(* LS Electric XG5000 project: 엘리베이터 프로젝트(내부 구현) *)
(* PLC LSPLC *)
(* module base 0 slot 0: FEnet:XGL-EFMT(B) (Fast Ethernet 통신 모듈, 전기 Master) *)
(* module base 0 slot 1: 입력 모듈:XGI-D21A (DC 24V 입력, 8점 (전류소스/싱크입력)) *)
(* module base 0 slot 2: 출력 모듈:XGQ-RY1A (릴레이 출력, 8점 (2A용, 단독 COM.)) *)
(* task 초기화: Kind=1 Priority=2 *)
VAR_GLOBAL
    ADD : INT;
    D0 : INT;
    D1 : INT;
    SUB : INT;
    열림TP : TP;
    타이머1 : TON;
END_VAR

(* Comments on direct variables
%MX0	상승
%MX1	하강
%MX2	문 열림
%MX3	문 닫힘
%MX4	도착
%MX5	비상 사태
%MX6	LOCK
%MX20	현재 1층 위치
%MX21	현재 2층 위치
%MX22	현재 3층 위치
%MX23	현재 4층 위치
%MX24	현재 5층 위치
%MX100	내부 1층 버튼
%MX101	내부2층버튼
%MX102	내부3층 버튼
%MX103	내부4층버튼
%MX104	내부5층버튼
%MX105	문열림 버튼
%MX106	문닫힘버튼
%MX107	외부1층상승
%MX108	외부 2층상승
%MX109	외부2층하강
%MX110	외부3층상승
%MX111	외부3층하강
%MX112	외부4층상승
%MX113	외부4층하강
%MX114	외부5층하강
%QX0.2.0	1층 램프
%QX0.2.1	2층 램프
%QX0.2.2	3층 램프
%QX0.2.3	4층 램프
%QX0.2.4	5층 램프
%QX0.2.5	문 열림
%QX0.2.6	문 닫힘
*)

PROGRAM 내부 (* task: 스캔 프로그램 *)
VAR_EXTERNAL
    D0 : INT;
    D1 : INT;
END_VAR
VAR
    D10 : INT;
    T2 : TON;
END_VAR
VAR
    _e1 : R_TRIG;
    _e2 : R_TRIG;
    _e3 : R_TRIG;
    _e4 : R_TRIG;
    _e5 : R_TRIG;
    _e6 : R_TRIG;
    _e7 : R_TRIG;
    _e8 : R_TRIG;
    _e9 : R_TRIG;
    _e10 : R_TRIG;
    _e11 : R_TRIG;
    _e12 : R_TRIG;
    _e13 : R_TRIG;
    _t14 : BOOL;
END_VAR

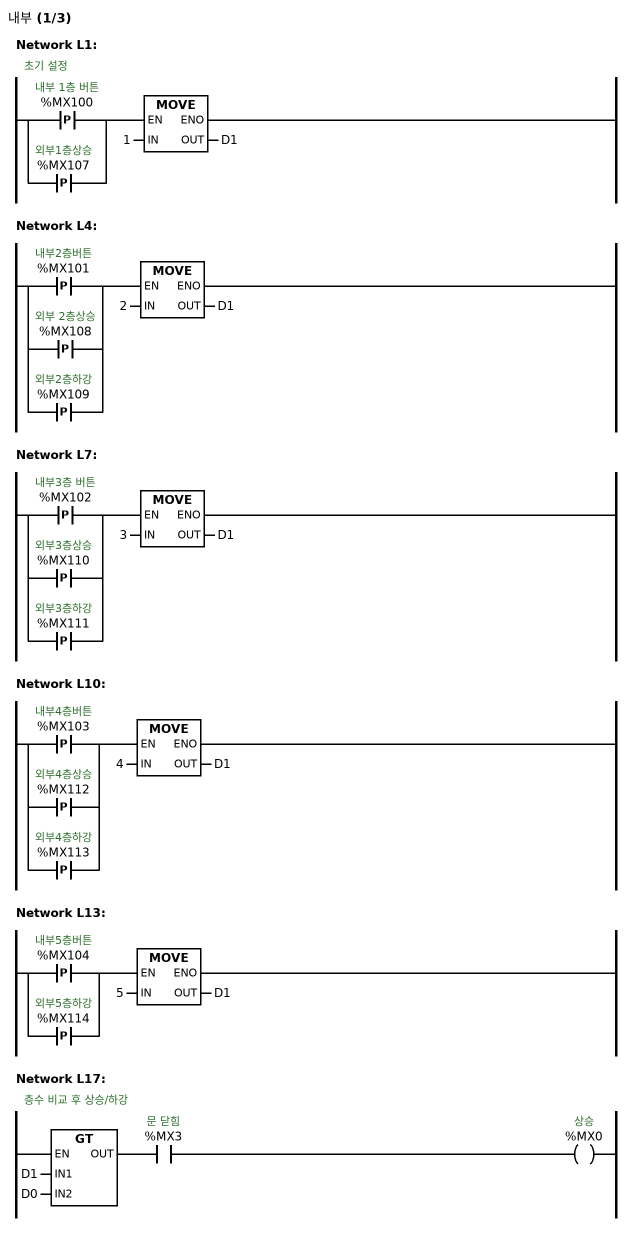
(* 초기 설정 *)
(* Rung L1 *)
_e1(CLK := %MX100);
_e2(CLK := %MX107);
IF _e1.Q OR _e2.Q THEN D1 := 1; END_IF;
(* Rung L4 *)
_e3(CLK := %MX101);
_e4(CLK := %MX108);
_e5(CLK := %MX109);
IF _e3.Q OR _e4.Q OR _e5.Q THEN D1 := 2; END_IF;
(* Rung L7 *)
_e6(CLK := %MX102);
_e7(CLK := %MX110);
_e8(CLK := %MX111);
IF _e6.Q OR _e7.Q OR _e8.Q THEN D1 := 3; END_IF;
(* Rung L10 *)
_e9(CLK := %MX103);
_e10(CLK := %MX112);
_e11(CLK := %MX113);
IF _e9.Q OR _e10.Q OR _e11.Q THEN D1 := 4; END_IF;
(* Rung L13 *)
_e12(CLK := %MX104);
_e13(CLK := %MX114);
IF _e12.Q OR _e13.Q THEN D1 := 5; END_IF;
(* 층수 비교 후 상승/하강 *)
(* Rung L17 *)
%MX0 := (D1 > D0) AND %MX3;

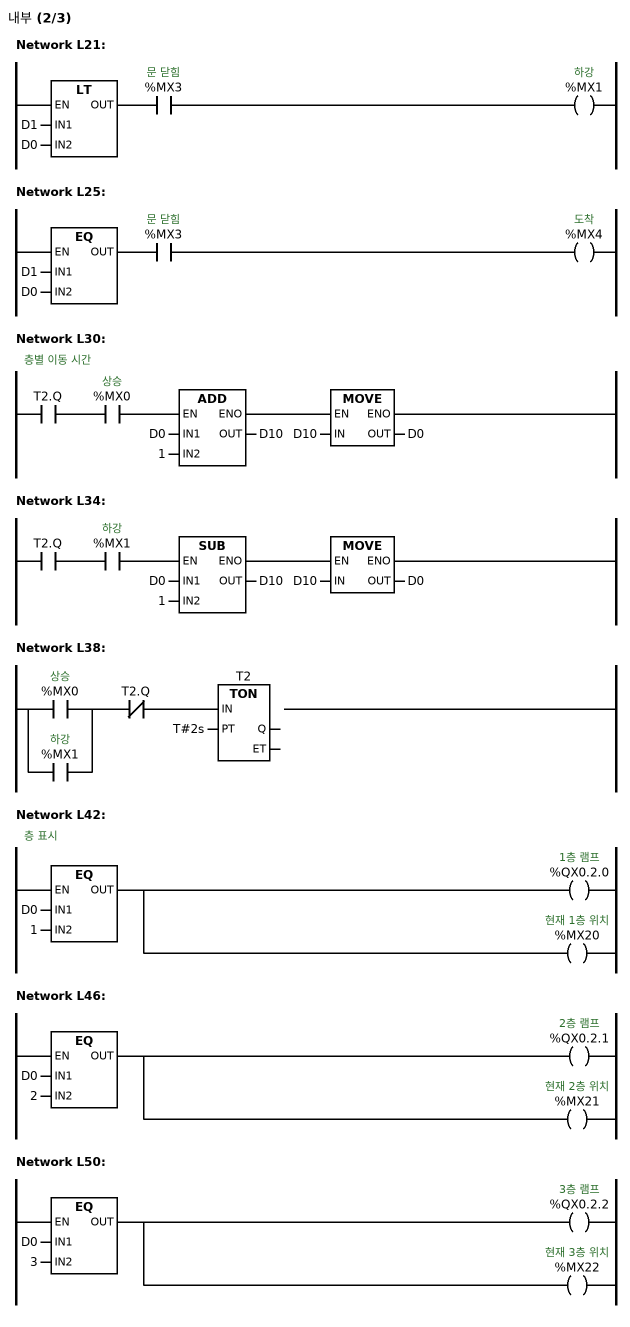
(* Rung L21 *)
%MX1 := (D1 < D0) AND %MX3;
(* Rung L25 *)
%MX4 := (D1 = D0) AND %MX3;
(* 층별 이동 시간 *)
(* Rung L30 *)
IF T2.Q AND %MX0 THEN
    D10 := D0 + 1;
    D0 := D10;
END_IF;
(* Rung L34 *)
IF T2.Q AND %MX1 THEN
    D10 := D0 - 1;
    D0 := D10;
END_IF;
(* Rung L38 *)
T2(IN := (%MX0 OR %MX1) AND NOT T2.Q, PT := T#2s);
(* 층 표시 *)
(* Rung L42 *)
%QX0.2.0 := D0 = 1;
%MX20 := D0 = 1;
(* Rung L46 *)
%QX0.2.1 := D0 = 2;
%MX21 := D0 = 2;
(* Rung L50 *)
%QX0.2.2 := D0 = 3;
%MX22 := D0 = 3;

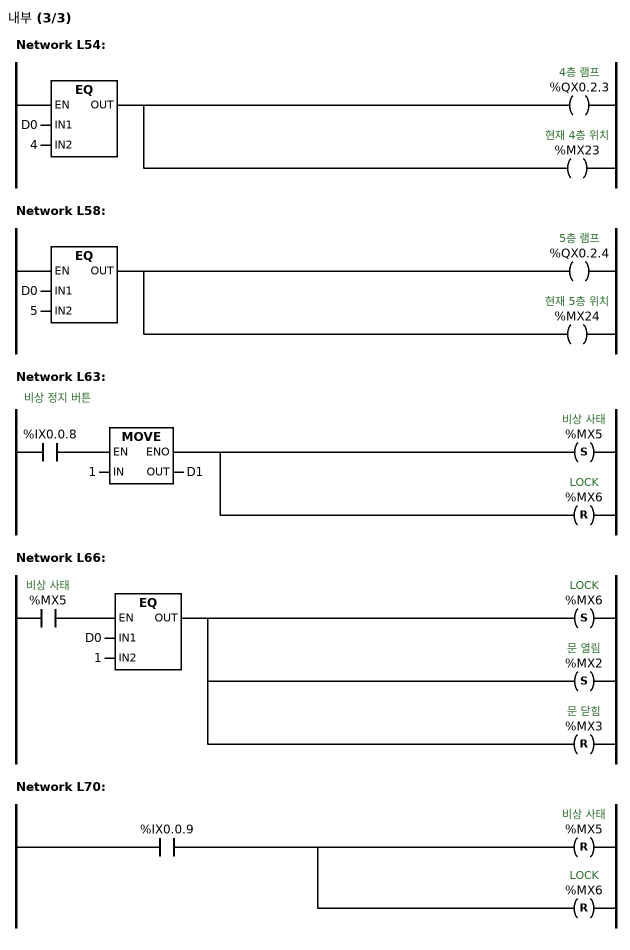
(* Rung L54 *)
%QX0.2.3 := D0 = 4;
%MX23 := D0 = 4;
(* Rung L58 *)
%QX0.2.4 := D0 = 5;
%MX24 := D0 = 5;
(* 비상 정지 버튼 *)
(* Rung L63 *)
IF %IX0.0.8 THEN
    D1 := 1;
    %MX5 := TRUE;
    %MX6 := FALSE;
END_IF;
(* Rung L66 *)
IF %MX5 THEN _t14 := D0 = 1; END_IF;
IF _t14 THEN
    %MX6 := TRUE;
    %MX2 := TRUE;
    %MX3 := FALSE;
END_IF;
(* Rung L70 *)
IF %IX0.0.9 THEN
    %MX5 := FALSE;
    %MX6 := FALSE;
END_IF;
END_PROGRAM

PROGRAM Timer (* task: 스캔 프로그램 *)
VAR
    CTU1 : CTU_INT;
    CTU2 : CTU_INT;
    D0 : SINT;
    OPEN : TP;
    T1 : TON;
    T2 : TON;
END_VAR
VAR_EXTERNAL
    열림TP : TP;
    타이머1 : TON;
END_VAR

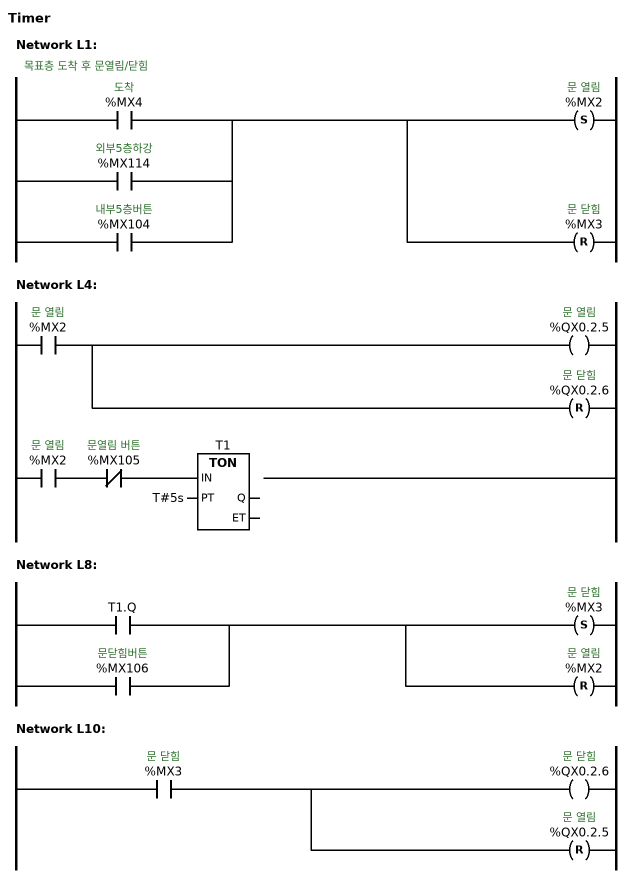
(* 목표층 도착 후 문열림/닫힘 *)
(* Rung L1 *)
IF %MX4 OR %MX114 OR %MX104 THEN
    %MX2 := TRUE;
    %MX3 := FALSE;
END_IF;
(* Rung L4 *)
%QX0.2.5 := %MX2;
IF %MX2 THEN %QX0.2.6 := FALSE; END_IF;
T1(IN := %MX2 AND NOT %MX105, PT := T#5s);
(* Rung L8 *)
IF T1.Q OR %MX106 THEN
    %MX3 := TRUE;
    %MX2 := FALSE;
END_IF;
(* Rung L10 *)
%QX0.2.6 := %MX3;
IF %MX3 THEN %QX0.2.5 := FALSE; END_IF;
END_PROGRAM

PROGRAM init (* task: 초기화 *)
VAR_EXTERNAL
    D0 : INT;
    D1 : INT;
END_VAR

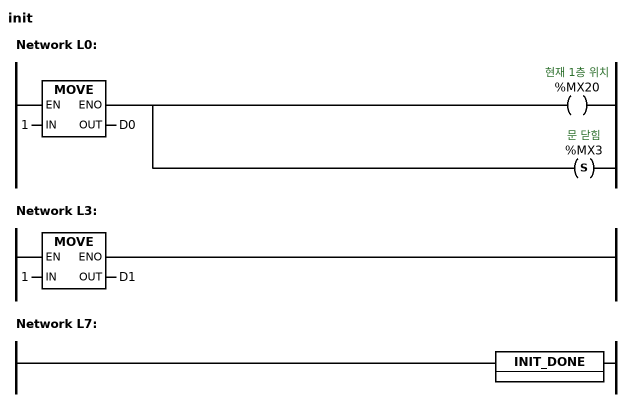
(* Rung L0 *)
D0 := 1;
%MX20 := TRUE;
%MX3 := TRUE;
(* Rung L3 *)
D1 := 1;
(* Rung L7 *)
INIT_DONE();
END_PROGRAM